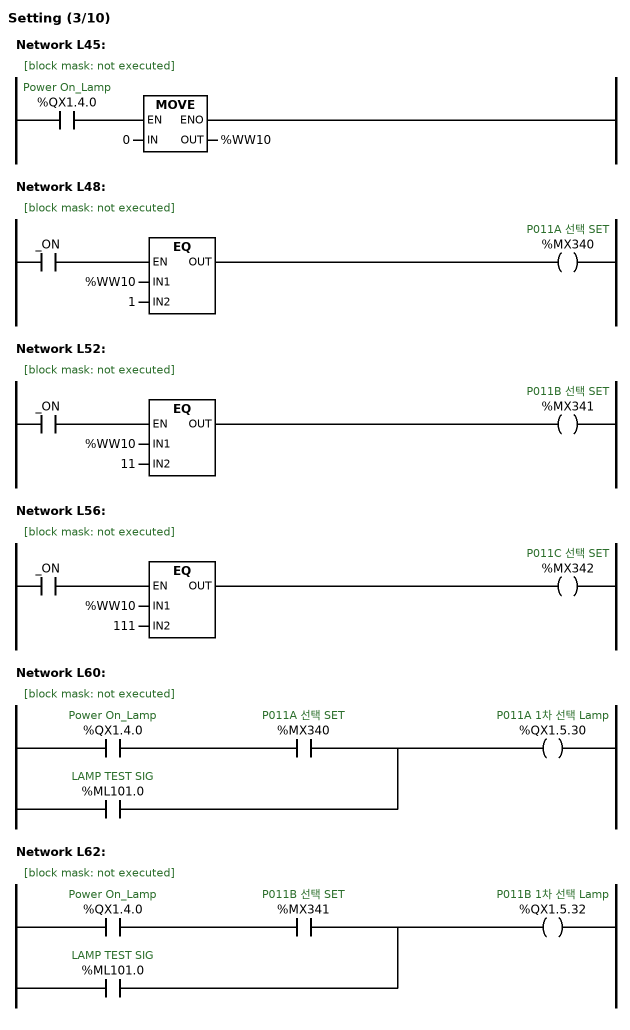
(* [picture p48: Setting rungs L45-L62] *)
(* Rung L45 is block-masked: not executed *)
// IF %QX1.4.0 THEN %WW10 := 0; END_IF;
(* Rung L48 is block-masked: not executed *)
// IF _ON THEN _t10 := %WW10 = 1; END_IF;
// %MX340 := _t10;
(* Rung L52 is block-masked: not executed *)
// IF _ON THEN _t11 := %WW10 = 11; END_IF;
// %MX341 := _t11;
(* Rung L56 is block-masked: not executed *)
// IF _ON THEN _t12 := %WW10 = 111; END_IF;
// %MX342 := _t12;
(* Rung L60 is block-masked: not executed *)
// %QX1.5.30 := (%QX1.4.0 AND %MX340) OR %ML101.0;
(* Rung L62 is block-masked: not executed *)
// %QX1.5.32 := (%QX1.4.0 AND %MX341) OR %ML101.0;

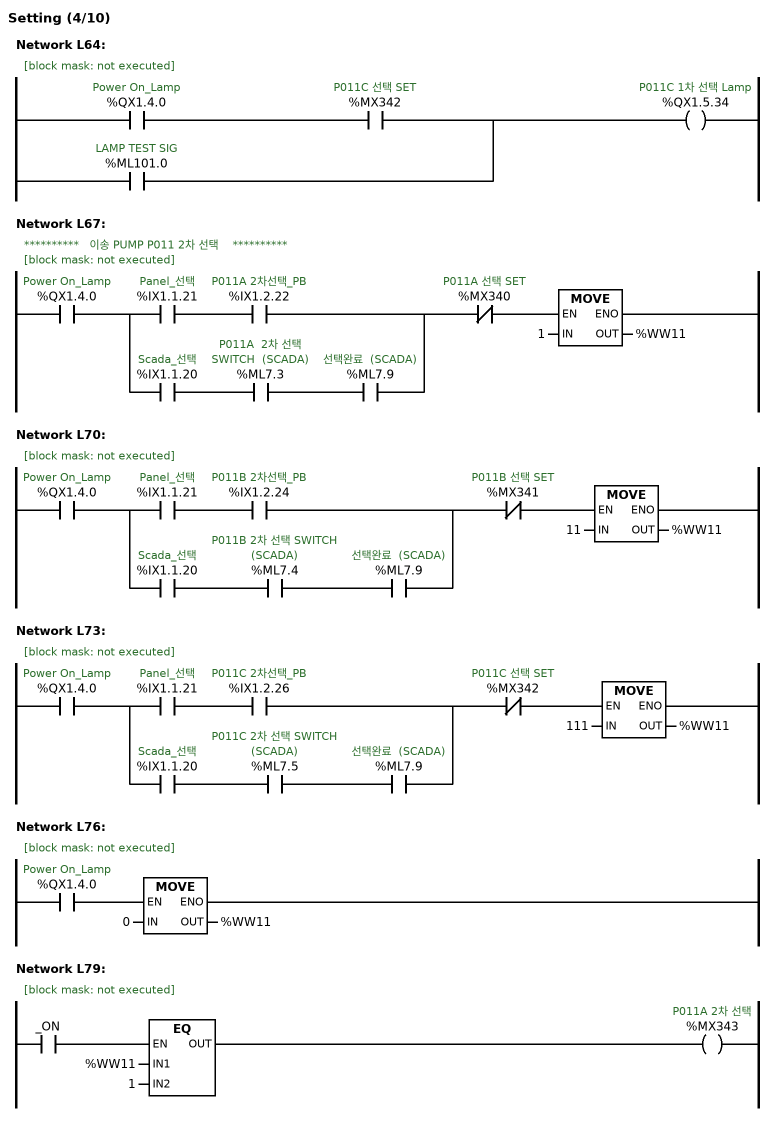
(* Rung L64 is block-masked: not executed *)
// %QX1.5.34 := (%QX1.4.0 AND %MX342) OR %ML101.0;
(* **********   이송 PUMP P011 2차 선택    ********** *)
(* Rung L67 is block-masked: not executed *)
// IF %QX1.4.0 AND ((%IX1.1.21 AND %IX1.2.22) OR (%IX1.1.20 AND %ML7.3 AND %ML7.9)) AND NOT %MX340 THEN
//     %WW11 := 1;
// END_IF;
(* Rung L70 is block-masked: not executed *)
// IF %QX1.4.0 AND ((%IX1.1.21 AND %IX1.2.24) OR (%IX1.1.20 AND %ML7.4 AND %ML7.9)) AND NOT %MX341 THEN
//     %WW11 := 11;
// END_IF;
(* Rung L73 is block-masked: not executed *)
// IF %QX1.4.0 AND ((%IX1.1.21 AND %IX1.2.26) OR (%IX1.1.20 AND %ML7.5 AND %ML7.9)) AND NOT %MX342 THEN
//     %WW11 := 111;
// END_IF;
(* Rung L76 is block-masked: not executed *)
// IF %QX1.4.0 THEN %WW11 := 0; END_IF;
(* Rung L79 is block-masked: not executed *)
// IF _ON THEN _t13 := %WW11 = 1; END_IF;
// %MX343 := _t13;

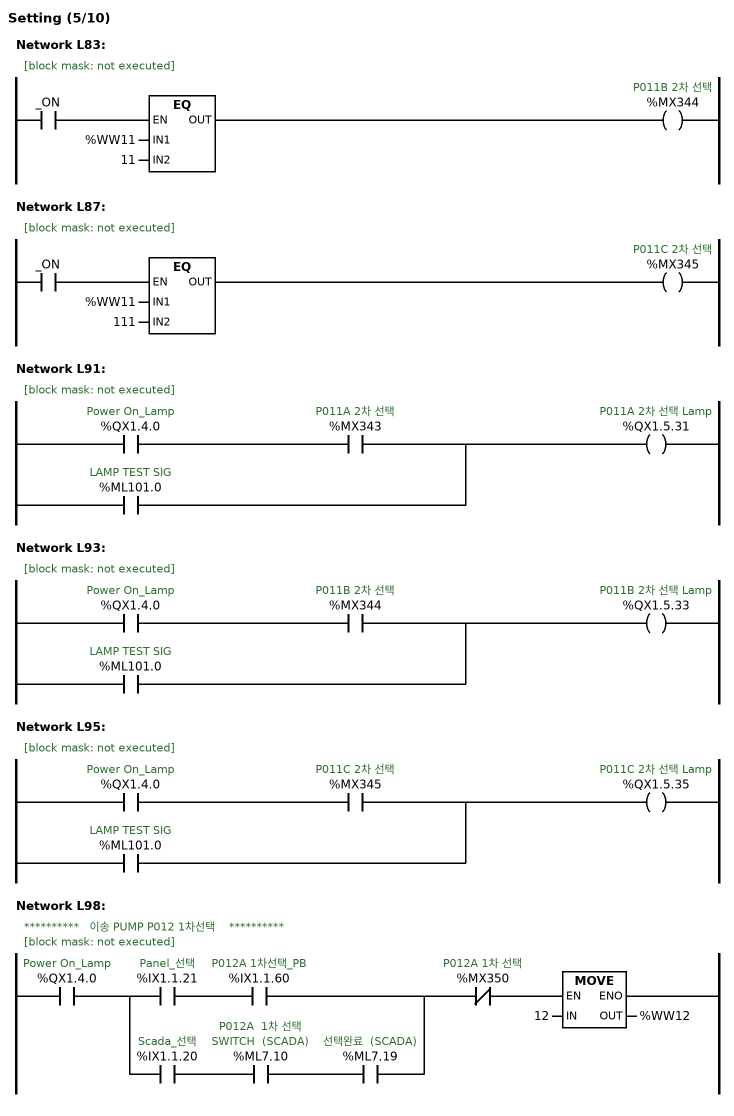
(* Rung L83 is block-masked: not executed *)
// IF _ON THEN _t14 := %WW11 = 11; END_IF;
// %MX344 := _t14;
(* Rung L87 is block-masked: not executed *)
// IF _ON THEN _t15 := %WW11 = 111; END_IF;
// %MX345 := _t15;
(* Rung L91 is block-masked: not executed *)
// %QX1.5.31 := (%QX1.4.0 AND %MX343) OR %ML101.0;
(* Rung L93 is block-masked: not executed *)
// %QX1.5.33 := (%QX1.4.0 AND %MX344) OR %ML101.0;
(* Rung L95 is block-masked: not executed *)
// %QX1.5.35 := (%QX1.4.0 AND %MX345) OR %ML101.0;
(* **********   이송 PUMP P012 1차선택    ********** *)
(* Rung L98 is block-masked: not executed *)
// IF %QX1.4.0 AND ((%IX1.1.21 AND %IX1.1.60) OR (%IX1.1.20 AND %ML7.10 AND %ML7.19)) AND NOT %MX350 THEN
//     %WW12 := 12;
// END_IF;

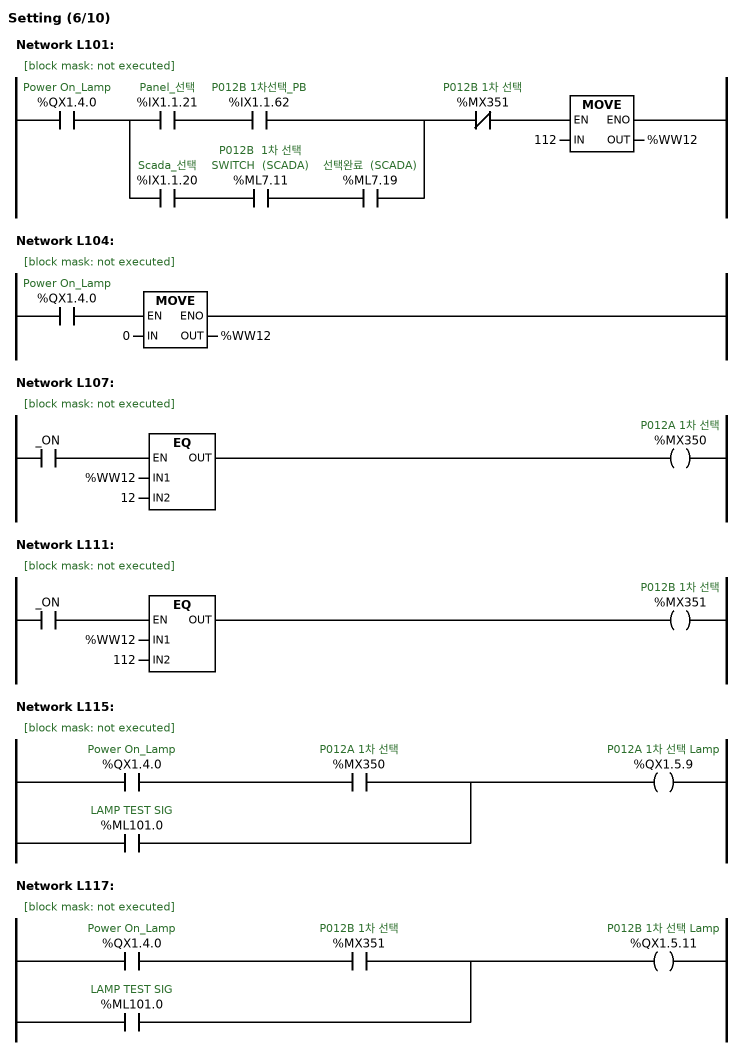
(* Rung L101 is block-masked: not executed *)
// IF %QX1.4.0 AND ((%IX1.1.21 AND %IX1.1.62) OR (%IX1.1.20 AND %ML7.11 AND %ML7.19)) AND NOT %MX351 THEN
//     %WW12 := 112;
// END_IF;
(* Rung L104 is block-masked: not executed *)
// IF %QX1.4.0 THEN %WW12 := 0; END_IF;
(* Rung L107 is block-masked: not executed *)
// IF _ON THEN _t16 := %WW12 = 12; END_IF;
// %MX350 := _t16;
(* Rung L111 is block-masked: not executed *)
// IF _ON THEN _t17 := %WW12 = 112; END_IF;
// %MX351 := _t17;
(* Rung L115 is block-masked: not executed *)
// %QX1.5.9 := (%QX1.4.0 AND %MX350) OR %ML101.0;
(* Rung L117 is block-masked: not executed *)
// %QX1.5.11 := (%QX1.4.0 AND %MX351) OR %ML101.0;

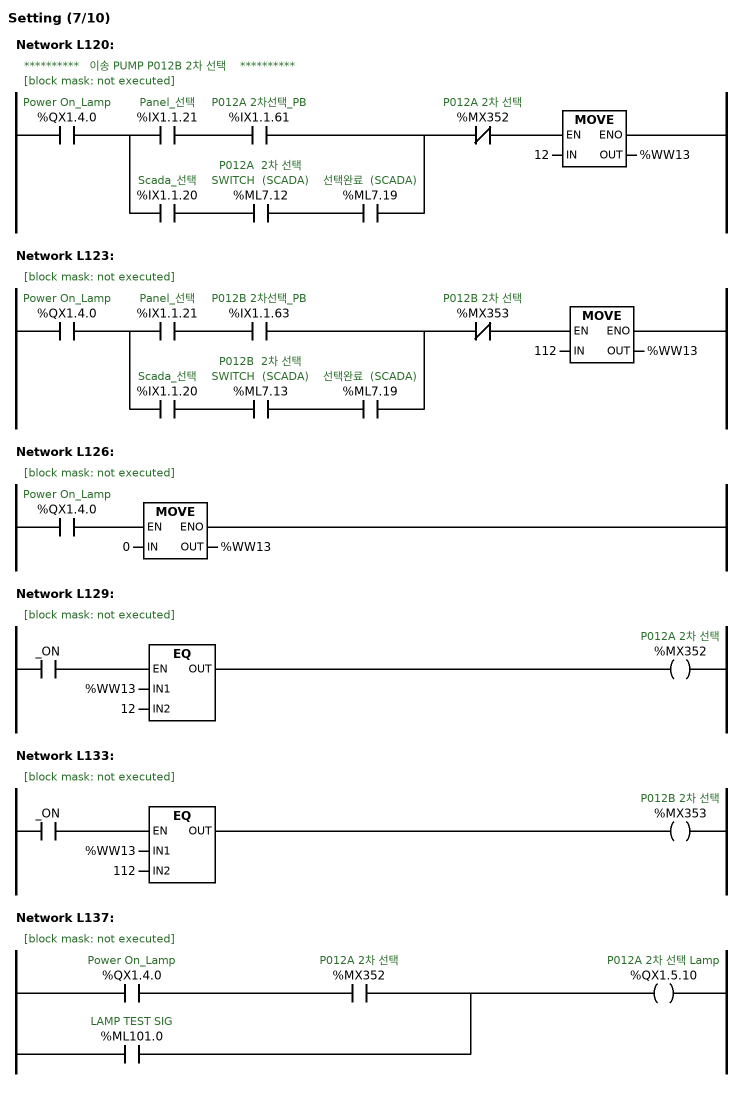
(* **********   이송 PUMP P012B 2차 선택    ********** *)
(* Rung L120 is block-masked: not executed *)
// IF %QX1.4.0 AND ((%IX1.1.21 AND %IX1.1.61) OR (%IX1.1.20 AND %ML7.12 AND %ML7.19)) AND NOT %MX352 THEN
//     %WW13 := 12;
// END_IF;
(* Rung L123 is block-masked: not executed *)
// IF %QX1.4.0 AND ((%IX1.1.21 AND %IX1.1.63) OR (%IX1.1.20 AND %ML7.13 AND %ML7.19)) AND NOT %MX353 THEN
//     %WW13 := 112;
// END_IF;
(* Rung L126 is block-masked: not executed *)
// IF %QX1.4.0 THEN %WW13 := 0; END_IF;
(* Rung L129 is block-masked: not executed *)
// IF _ON THEN _t18 := %WW13 = 12; END_IF;
// %MX352 := _t18;
(* Rung L133 is block-masked: not executed *)
// IF _ON THEN _t19 := %WW13 = 112; END_IF;
// %MX353 := _t19;
(* Rung L137 is block-masked: not executed *)
// %QX1.5.10 := (%QX1.4.0 AND %MX352) OR %ML101.0;

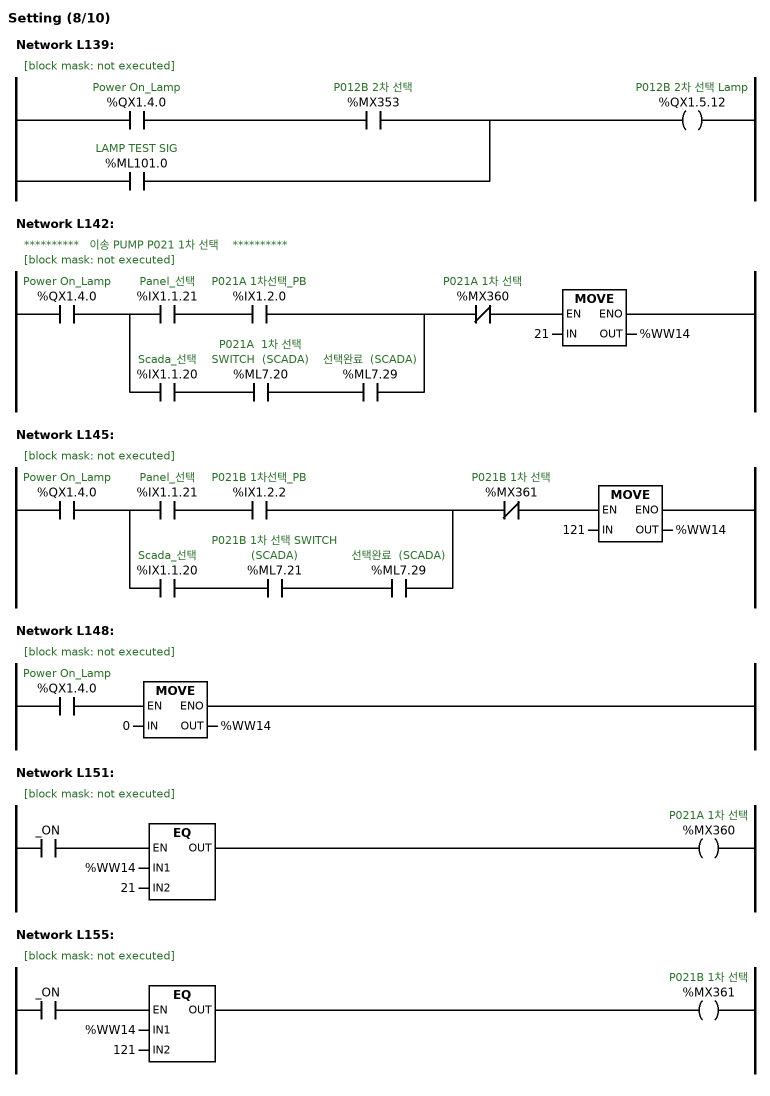
(* Rung L139 is block-masked: not executed *)
// %QX1.5.12 := (%QX1.4.0 AND %MX353) OR %ML101.0;
(* **********   이송 PUMP P021 1차 선택    ********** *)
(* Rung L142 is block-masked: not executed *)
// IF %QX1.4.0 AND ((%IX1.1.21 AND %IX1.2.0) OR (%IX1.1.20 AND %ML7.20 AND %ML7.29)) AND NOT %MX360 THEN
//     %WW14 := 21;
// END_IF;
(* Rung L145 is block-masked: not executed *)
// IF %QX1.4.0 AND ((%IX1.1.21 AND %IX1.2.2) OR (%IX1.1.20 AND %ML7.21 AND %ML7.29)) AND NOT %MX361 THEN
//     %WW14 := 121;
// END_IF;
(* Rung L148 is block-masked: not executed *)
// IF %QX1.4.0 THEN %WW14 := 0; END_IF;
(* Rung L151 is block-masked: not executed *)
// IF _ON THEN _t20 := %WW14 = 21; END_IF;
// %MX360 := _t20;
(* Rung L155 is block-masked: not executed *)
// IF _ON THEN _t21 := %WW14 = 121; END_IF;
// %MX361 := _t21;

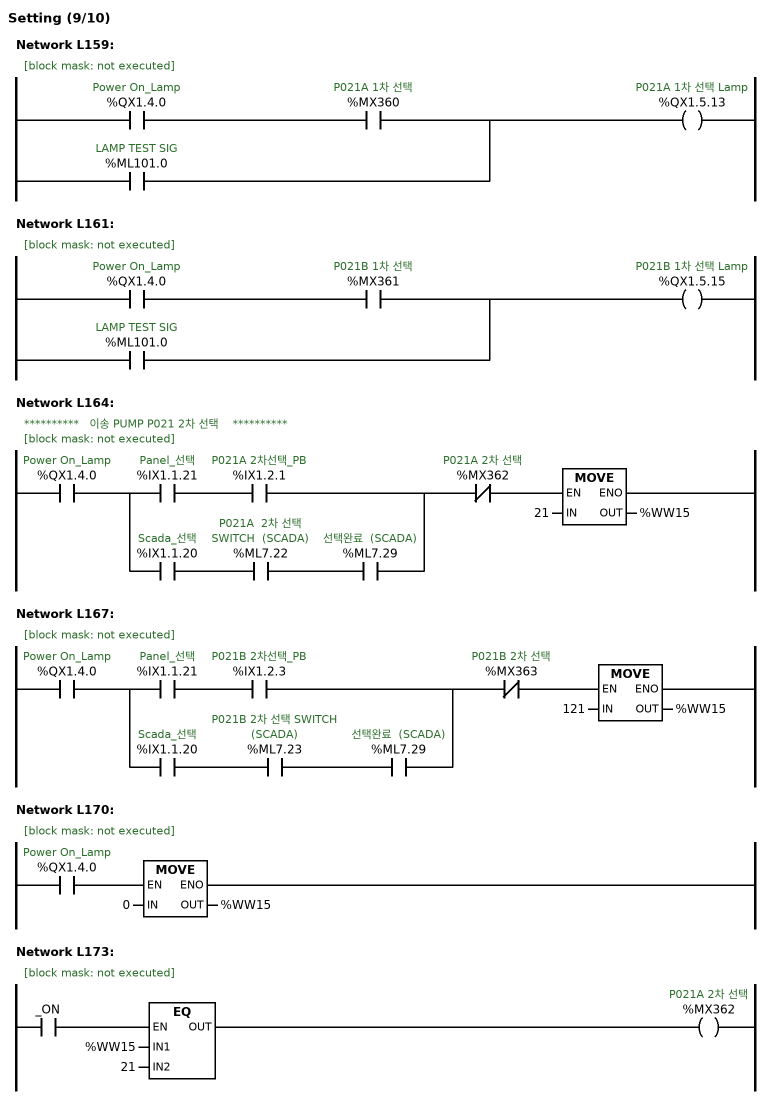
(* Rung L159 is block-masked: not executed *)
// %QX1.5.13 := (%QX1.4.0 AND %MX360) OR %ML101.0;
(* Rung L161 is block-masked: not executed *)
// %QX1.5.15 := (%QX1.4.0 AND %MX361) OR %ML101.0;
(* **********   이송 PUMP P021 2차 선택    ********** *)
(* Rung L164 is block-masked: not executed *)
// IF %QX1.4.0 AND ((%IX1.1.21 AND %IX1.2.1) OR (%IX1.1.20 AND %ML7.22 AND %ML7.29)) AND NOT %MX362 THEN
//     %WW15 := 21;
// END_IF;
(* Rung L167 is block-masked: not executed *)
// IF %QX1.4.0 AND ((%IX1.1.21 AND %IX1.2.3) OR (%IX1.1.20 AND %ML7.23 AND %ML7.29)) AND NOT %MX363 THEN
//     %WW15 := 121;
// END_IF;
(* Rung L170 is block-masked: not executed *)
// IF %QX1.4.0 THEN %WW15 := 0; END_IF;
(* Rung L173 is block-masked: not executed *)
// IF _ON THEN _t22 := %WW15 = 21; END_IF;
// %MX362 := _t22;

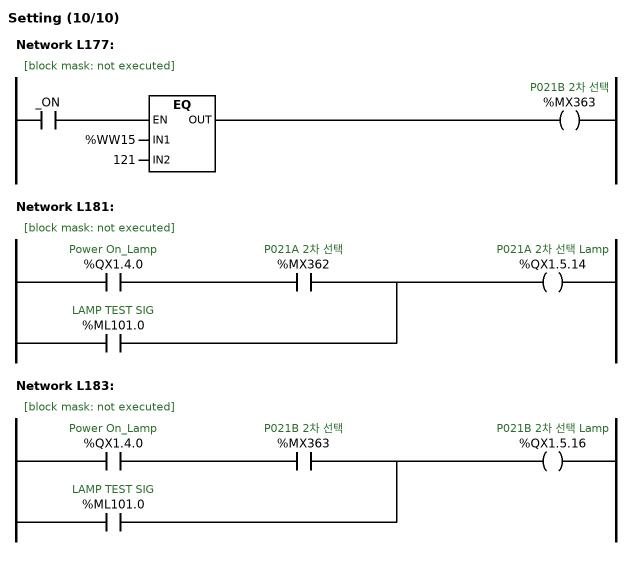
(* Rung L177 is block-masked: not executed *)
// IF _ON THEN _t23 := %WW15 = 121; END_IF;
// %MX363 := _t23;
(* Rung L181 is block-masked: not executed *)
// %QX1.5.14 := (%QX1.4.0 AND %MX362) OR %ML101.0;
(* Rung L183 is block-masked: not executed *)
// %QX1.5.16 := (%QX1.4.0 AND %MX363) OR %ML101.0;
END_PROGRAM

PROGRAM Alarm (* task: 스캔 프로그램 *)

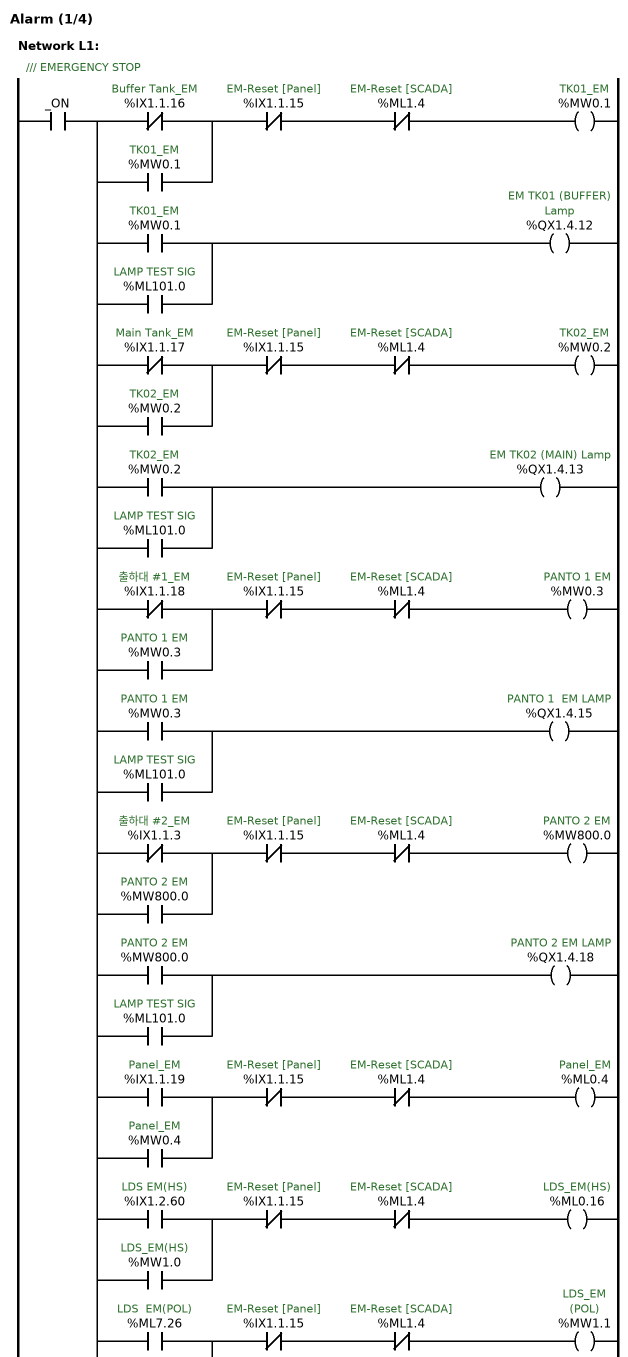

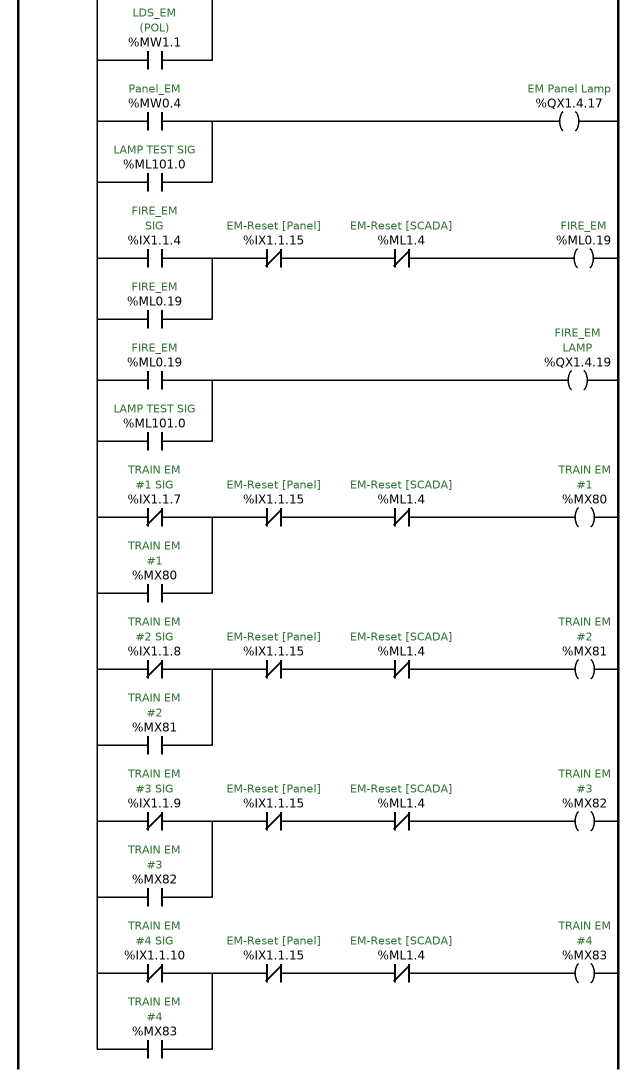
(* /// EMERGENCY STOP *)
(* Rung L1 *)
%MW0.1 := _ON AND (NOT %IX1.1.16 OR %MW0.1) AND NOT %IX1.1.15 AND NOT %ML1.4;
%QX1.4.12 := _ON AND (%MW0.1 OR %ML101.0);
%MW0.2 := _ON AND (NOT %IX1.1.17 OR %MW0.2) AND NOT %IX1.1.15 AND NOT %ML1.4;
%QX1.4.13 := _ON AND (%MW0.2 OR %ML101.0);
%MW0.3 := _ON AND (NOT %IX1.1.18 OR %MW0.3) AND NOT %IX1.1.15 AND NOT %ML1.4;
%QX1.4.15 := _ON AND (%MW0.3 OR %ML101.0);
%MW800.0 := _ON AND (NOT %IX1.1.3 OR %MW800.0) AND NOT %IX1.1.15 AND NOT %ML1.4;
%QX1.4.18 := _ON AND (%MW800.0 OR %ML101.0);
%ML0.4 := _ON AND (%IX1.1.19 OR %MW0.4) AND NOT %IX1.1.15 AND NOT %ML1.4;
%ML0.16 := _ON AND (%IX1.2.60 OR %MW1.0) AND NOT %IX1.1.15 AND NOT %ML1.4;
%MW1.1 := _ON AND (%ML7.26 OR %MW1.1) AND NOT %IX1.1.15 AND NOT %ML1.4;
%QX1.4.17 := _ON AND (%MW0.4 OR %ML101.0);
%ML0.19 := _ON AND (%IX1.1.4 OR %ML0.19) AND NOT %IX1.1.15 AND NOT %ML1.4;
%QX1.4.19 := _ON AND (%ML0.19 OR %ML101.0);
%MX80 := _ON AND (NOT %IX1.1.7 OR %MX80) AND NOT %IX1.1.15 AND NOT %ML1.4;
%MX81 := _ON AND (NOT %IX1.1.8 OR %MX81) AND NOT %IX1.1.15 AND NOT %ML1.4;
%MX82 := _ON AND (NOT %IX1.1.9 OR %MX82) AND NOT %IX1.1.15 AND NOT %ML1.4;
%MX83 := _ON AND (NOT %IX1.1.10 OR %MX83) AND NOT %IX1.1.15 AND NOT %ML1.4;

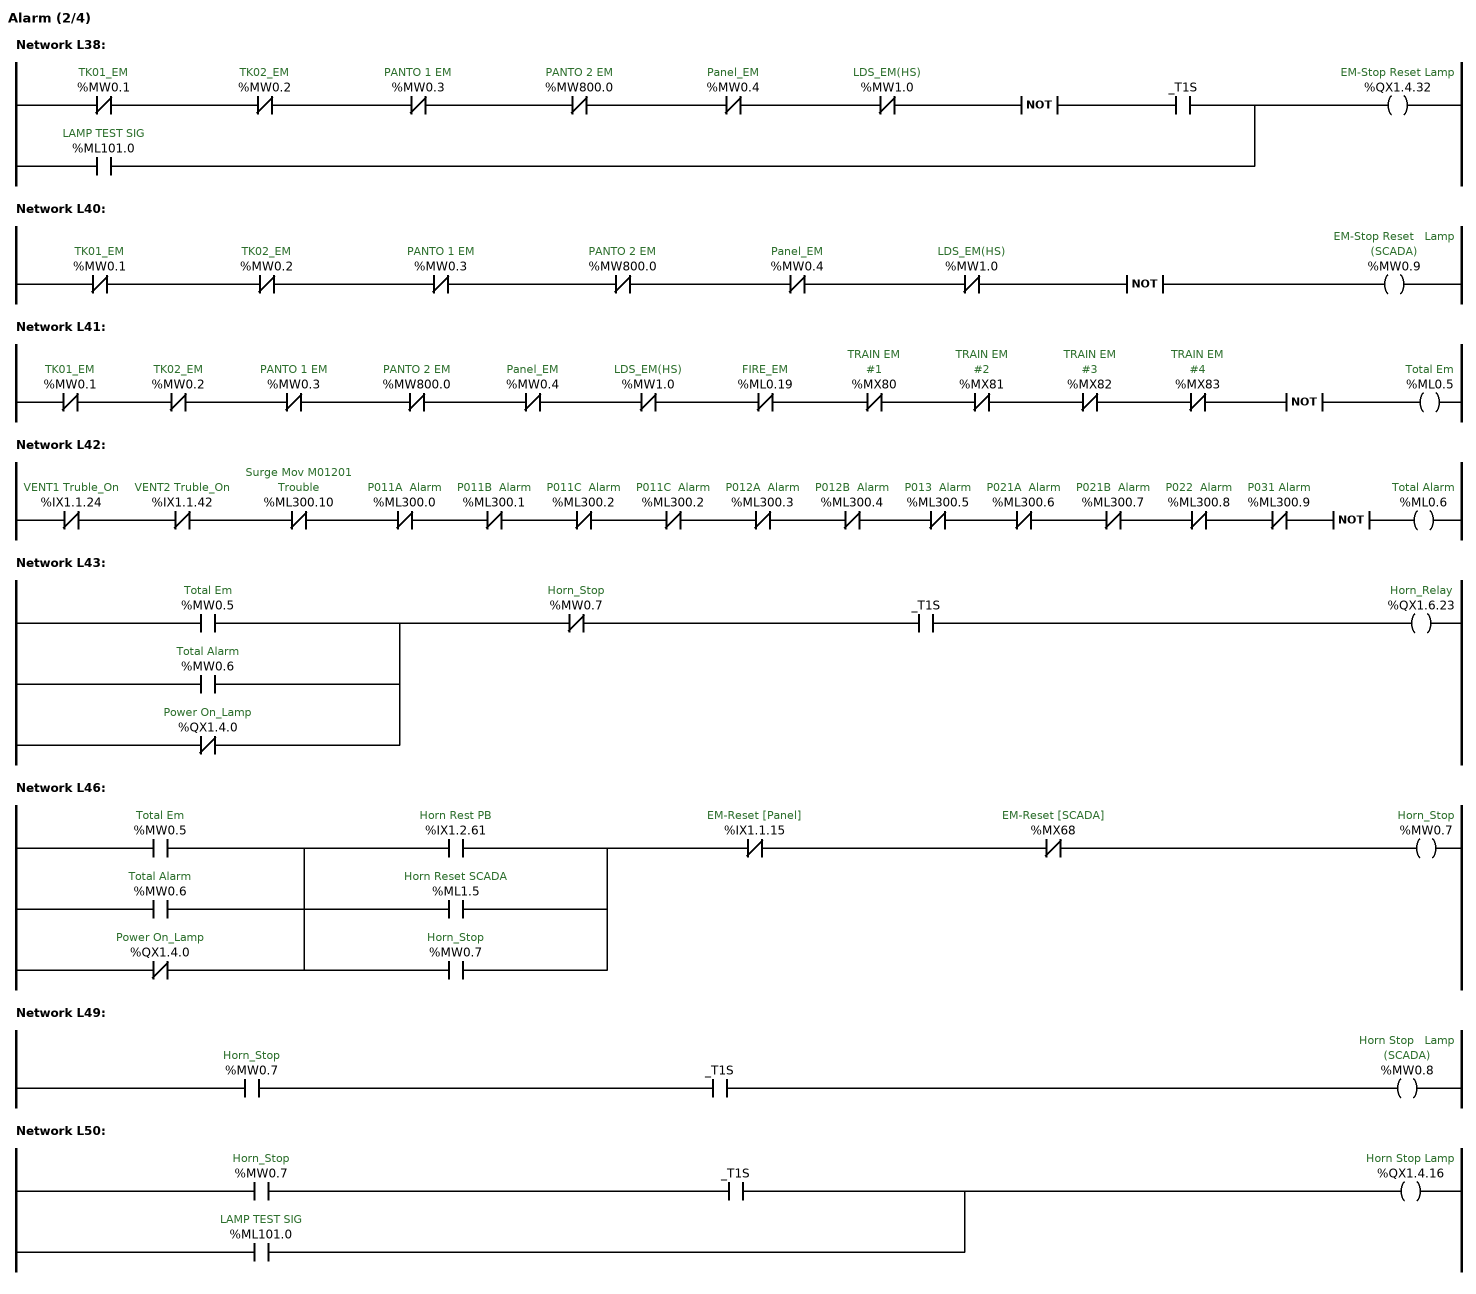
(* Rung L38 *)
%QX1.4.32 := (NOT (NOT %MW0.1 AND NOT %MW0.2 AND NOT %MW0.3 AND NOT %MW800.0 AND NOT %MW0.4 AND NOT %MW1.0) AND _T1S) OR %ML101.0;
(* Rung L40 *)
%MW0.9 := NOT (NOT %MW0.1 AND NOT %MW0.2 AND NOT %MW0.3 AND NOT %MW800.0 AND NOT %MW0.4 AND NOT %MW1.0);
(* Rung L41 *)
%ML0.5 := NOT (NOT %MW0.1 AND NOT %MW0.2 AND NOT %MW0.3 AND NOT %MW800.0 AND NOT %MW0.4 AND NOT %MW1.0 AND NOT %ML0.19 AND NOT %MX80 AND NOT %MX81 AND NOT %MX82 AND NOT %MX83);
(* Rung L42 *)
%ML0.6 := NOT (NOT %IX1.1.24 AND NOT %IX1.1.42 AND NOT %ML300.10 AND NOT %ML300.0 AND NOT %ML300.1 AND NOT %ML300.2 AND NOT %ML300.2 AND NOT %ML300.3 AND NOT %ML300.4 AND NOT %ML300.5 AND NOT %ML300.6 AND NOT %ML300.7 AND NOT %ML300.8 AND NOT %ML300.9);
(* Rung L43 *)
%QX1.6.23 := (%MW0.5 OR %MW0.6 OR NOT %QX1.4.0) AND NOT %MW0.7 AND _T1S;
(* Rung L46 *)
%MW0.7 := (%MW0.5 OR %MW0.6 OR NOT %QX1.4.0) AND (%IX1.2.61 OR %ML1.5 OR %MW0.7) AND NOT %IX1.1.15 AND NOT %MX68;
(* Rung L49 *)
%MW0.8 := %MW0.7 AND _T1S;
(* Rung L50 *)
%QX1.4.16 := (%MW0.7 AND _T1S) OR %ML101.0;

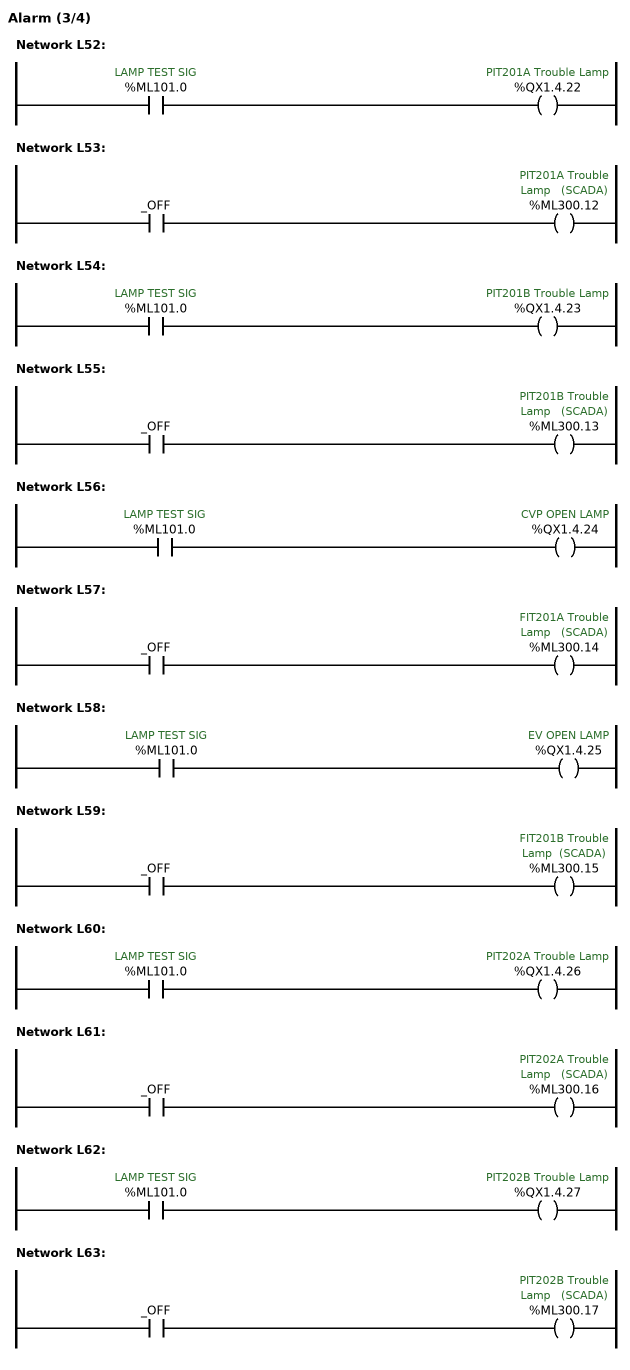
(* Rung L52 *)
%QX1.4.22 := %ML101.0;
(* Rung L53 *)
%ML300.12 := _OFF;
(* Rung L54 *)
%QX1.4.23 := %ML101.0;
(* Rung L55 *)
%ML300.13 := _OFF;
(* Rung L56 *)
%QX1.4.24 := %ML101.0;
(* Rung L57 *)
%ML300.14 := _OFF;
(* Rung L58 *)
%QX1.4.25 := %ML101.0;
(* Rung L59 *)
%ML300.15 := _OFF;
(* Rung L60 *)
%QX1.4.26 := %ML101.0;
(* Rung L61 *)
%ML300.16 := _OFF;
(* Rung L62 *)
%QX1.4.27 := %ML101.0;
(* Rung L63 *)
%ML300.17 := _OFF;

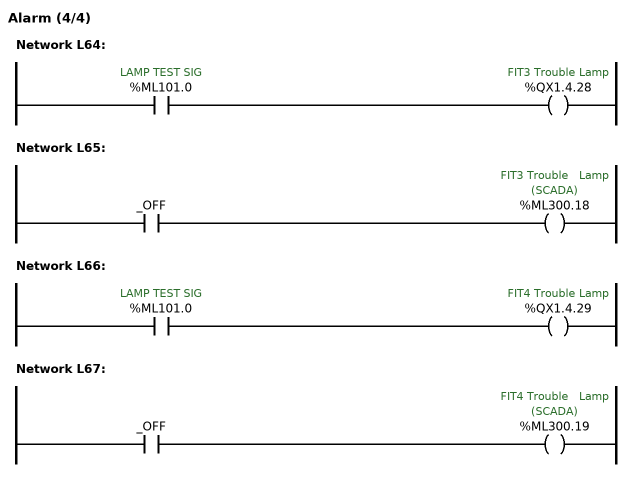
(* Rung L64 *)
%QX1.4.28 := %ML101.0;
(* Rung L65 *)
%ML300.18 := _OFF;
(* Rung L66 *)
%QX1.4.29 := %ML101.0;
(* Rung L67 *)
%ML300.19 := _OFF;
END_PROGRAM